ABB RobotStudio station: miniproject_v1_20180422-121856.rsstn

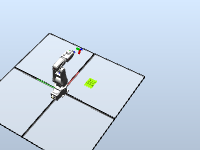
Station Station (saved by RobotStudio 6.6.7701.1025)
Controller miniproject
  mechanical unit ROB_1: IRB120_3_58__01, 6 joints, base frame (0, 0, 0) mm
Layout (positions relative to the parent item):
  - IRB120_3_58__01 [mechanism, from Robots\IRB120_3_58_G_01.rslib] at (0, 0, 0) mm; joint values [0, 0, 0, 0, 0.5236, 0] (rad or m)
  - Deliver plate 16x16 LEGO Plate [part] at (400, -300, 0) mm
  - lego2x2 Orange [part] at (329.44, -60.46, 0) mm, rotated rx 90 ry 0 rz 0 deg
  - lego2x2 Red [part] at (418.33, -49.7, 0) mm, rotated rx 90 ry 0 rz 0 deg
  - lego2x2 Yellow [part] at (549.33, 43.86, 0) mm, rotated rx 90 ry 0 rz 0 deg
  - lego2x2 Blue [part] at (490.71, 5.14, 0) mm, rotated rx 90 ry 0 rz 10 deg
  - lego2x2 Green [part] at (349.13, -4.15, 0) mm, rotated rx 90 ry 0 rz 80 deg
  - lego2x2 Blue [part] at (400.47, -14.74, 0) mm, rotated rx 90 ry 0 rz -26 deg
  - lego2x2 Blue_2 [part] at (381.32, -147, 0) mm, rotated rx 90 ry 0 rz 0 deg
  - lego2x2 Blue_3 [part] at (447.97, -80.48, 0) mm, rotated rx 90 ry 0 rz 15 deg
  - lego2x2 Blue_4 [part] at (370.2, -57.47, 0) mm, rotated rx 90 ry 0 rz 0 deg
  - lego2x2 Green_2 [part] at (457.03, -35.41, 0) mm, rotated rx 90 ry 0 rz 0 deg
  - lego2x2 Green_3 [part] at (450.9, 39.8, 0) mm, rotated rx 90 ry 0 rz 0 deg
  - lego2x2 Green_4 [part] at (395.13, 41.77, 0) mm, rotated rx 90 ry 0 rz -16 deg
  - lego2x2 Orange [part] at (387.07, -83.22, 0) mm, rotated rx 90 ry 0 rz -40 deg
  - lego2x2 Orange_2 [part] at (514.18, -61.46, 0) mm, rotated rx 90 ry 0 rz 0 deg
  - lego2x2 Orange_3 [part] at (542.01, -7.45, 0) mm, rotated rx 90 ry 0 rz -35 deg
  - lego2x2 Orange_4 [part] at (488.39, 78.35, 0) mm, rotated rx 90 ry 0 rz 0 deg
  - lego2x2 Yellow [part] at (427.89, -100.2, 0) mm, rotated rx 90 ry 0 rz -7 deg
  - lego2x2 Yellow_2 [part] at (498.8, -138.52, 0) mm, rotated rx 90 ry 0 rz 0 deg
  - lego2x2 Yellow_3 [part] at (447.5, 98.13, 0) mm, rotated rx 90 ry 0 rz -10 deg
  - lego2x2 Yellow_4 [part] at (361.28, 75.07, 0) mm, rotated rx 90 ry 0 rz 0 deg
  - lego2x2 Yellow_5 [part] at (286.67, -13.02, 0) mm, rotated rx 90 ry 0 rz 50 deg
  - lego2x2 Red [part] at (478.59, -79.86, 0) mm, rotated rx 90 ry 0 rz 0 deg
  - lego2x2 Red_2 [part] at (460.14, -3.62, 0) mm, rotated rx 90 ry 0 rz 17 deg
  - lego2x2 Red_3 [part] at (410.79, 82.14, 0) mm, rotated rx 90 ry 0 rz 0 deg
  - lego2x2 Red_4 [part] at (332.23, 31.54, 0) mm, rotated rx 90 ry 0 rz 35 deg
Targets, tools, work objects and paths stored in the station, written as RAPID:
! task T_ROB1
MODULE FunctionHandler
  PERS tooldata defaultTool:=[TRUE,[[0,0,0],[1,0,0,0]],[1,[0,0,0.001],[1,0,0,0],0,0,0]];
  PERS wobjdata defaultWobj:=[FALSE,TRUE,"",[[0,0,0],[1,0,0,0]],[[0,0,0],[1,0,0,0]]];
  VAR signaldo defaultTakePictureActivationIO;
  VAR signaldi defaultTakePictureExecutedIO;
  PROC FH_TakePicture()
    SetDO defaultTakePictureActivationIO,1;
    WaitDI defaultTakePictureExecutedIO,1;
    SetDO defaultTakePictureActivationIO,0;
  ENDPROC
ENDMODULE

! task T_ROB1
MODULE CommandHandler
  PROC COMH_CommandListener()
  ENDPROC
ENDMODULE

! task T_ROB1
MODULE Module1
  PROC main()
    IP_Initialize;
    COMH_CommandListener;
  ENDPROC
ENDMODULE

! task T_ROB1
MODULE InitParameters
  PROC IP_Initialize()
    ConfL \Off;
    ConfJ \Off;
  ENDPROC
ENDMODULE

! task T_ROB1
MODULE CalibData
  PERS tooldata SCHINK_WSG_GRIPPER_TOOL:=[TRUE,[[0,0,234.82],[1,0,0,0]],[5,[0,0,100],[1,0,0,0],0,0,0]];
ENDMODULE

